(* IEC 61131-3 sources: volt/packages/volt-lsp-iec/test-corpus/pro2193/Device/Plc Logic/Application, 1 file *)

(* ---- GVL_ComponentHardwareCall.pou ---- *)
{attribute 'linkalways'}
PROGRAM GVL_ComponentHardwareCall
VAR
END_VAR
%LANGUAGE ST
(* This code is generated automatically *)
(* Don't change the content! *)

//Controller
GVL_ComponentHardware.Device();

//EtherCAT device
GVL_ComponentHardware.L_i750_ZR();
GVL_ComponentHardware.L_i750_C2();
GVL_ComponentHardware.L_i750_M1();
GVL_ComponentHardware.L_i750_M2();
GVL_ComponentHardware.L_i750_Z();
GVL_ComponentHardware.L_i750_C1();
GVL_ComponentHardware.L_i750_Xi();
GVL_ComponentHardware.L_i750_Xu();
GVL_ComponentHardware.L_i950_Y();
GVL_ComponentHardware.RIO_M1();
GVL_ComponentHardware.RIO_Z1();
GVL_ComponentHardware.RIO_BFU();
GVL_ComponentHardware.FANUC_R_30iB_Plus();

//I/O module
GVL_ComponentHardware.DI_30();
GVL_ComponentHardware.DI_31();
GVL_ComponentHardware.DI_32();
GVL_ComponentHardware.DI_33();
GVL_ComponentHardware.DQ_30();
GVL_ComponentHardware.DQ_31();
GVL_ComponentHardware.DQ_32();
GVL_ComponentHardware.DQ_33();
GVL_ComponentHardware.DQ_34();
GVL_ComponentHardware.DQ_35();
GVL_ComponentHardware.DQ_36();
GVL_ComponentHardware.DI_40();
GVL_ComponentHardware.DI_41();
GVL_ComponentHardware.DI_42();
GVL_ComponentHardware.DI_43();
GVL_ComponentHardware.DI_44();
GVL_ComponentHardware.DI_45();
GVL_ComponentHardware.DQ_40();
GVL_ComponentHardware.DQ_41();
GVL_ComponentHardware.DQ_42();
GVL_ComponentHardware.DQ_43();
GVL_ComponentHardware.DQ_44();
GVL_ComponentHardware.DQ_45();
GVL_ComponentHardware.DQ_46();
GVL_ComponentHardware.DI_50();
GVL_ComponentHardware.DI_51();
GVL_ComponentHardware.DI_52();
GVL_ComponentHardware.DI_53();
GVL_ComponentHardware.DI_54();
GVL_ComponentHardware.DQ_50();
GVL_ComponentHardware.DQ_51();
GVL_ComponentHardware.DQ_52();
GVL_ComponentHardware.DQ_53();
GVL_ComponentHardware.DQ_54();

END_PROGRAM
